// TIA Portal V19 export
TYPE "FCP_IN"
   STRUCT
      EFCStatusWord { S7_SetPoint := 'True'} : "EFC_STATUS_WORD";
      EFCExStatusWord { S7_SetPoint := 'True'} : "EFC_EX_STATUS_WORD";
      FcPStatusWord { S7_SetPoint := 'True'} : "FCP_STATUS_WORD";
      SpeedAct : Word;
      PressureAct : Word;
      CurrentAct : Word;
      ASFWarningCode : Word;
      ASFErrorCode : Word;
   END_STRUCT;
END_TYPE
